// Mitsubishi GX Works2 project: 퀴즈쇼 부저 예제(인터록, 자기유지)   PLC: Q03UDV

PROGRAM MAIN
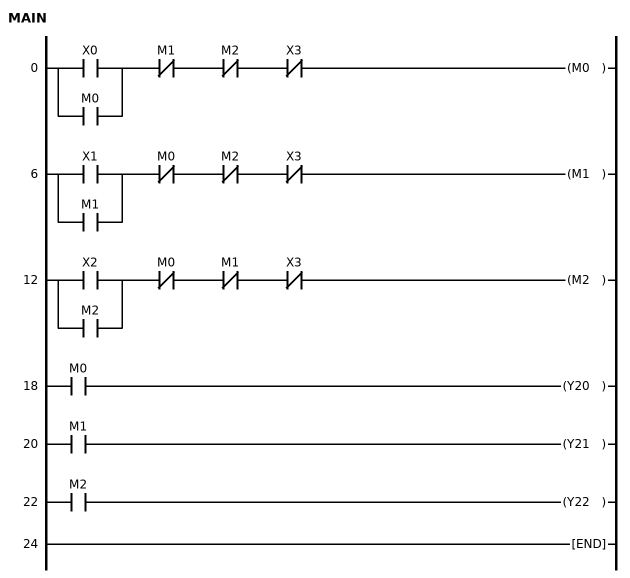
0     LD      X0
      OR      M0
      ANI     M1
      ANI     M2
      ANI     X3
      OUT     M0
6     LD      X1
      OR      M1
      ANI     M0
      ANI     M2
      ANI     X3
      OUT     M1
12    LD      X2
      OR      M2
      ANI     M0
      ANI     M1
      ANI     X3
      OUT     M2
18    LD      M0
      OUT     Y20
20    LD      M1
      OUT     Y21
22    LD      M2
      OUT     Y22
24    END
END_PROGRAM
